// TIA Portal V18 export
VAR_GLOBAL   // PLC tag table "04_7 Costanti Nomi Attuatore Stz07"
END_VAR
VAR_GLOBAL CONSTANT   // user constants
   M201 : Int := 1;   // Motore alimentatore
   P701 : Int := 2;   // EV Salita/discesa alimentatore
   "P01-01" : Int := 3;   // EV Cassetto stampo pressa
END_VAR
